FUNCTION_BLOCK FB_TaskMoveZ_creator IMPLEMENTS InterfaceTaskCreator
VAR_INPUT
END_VAR
VAR_OUTPUT
END_VAR
VAR
	_p				: MC_LREAL;
	_v				: MC_LREAL;
	_a				: MC_LREAL;
	_d				: MC_LREAL;
	_j				: MC_LREAL;
	_mover			: REFERENCE TO MC_PlanarMover;
END_VAR

{warning 'add method implementation '}
METHOD create_future : jobmgmt.InterfaceFuture
VAR_INPUT
	future_name	: STRING;
END_VAR
VAR
	_p_future : POINTER TO FB_TaskMoveZ;
END_VAR
_p_future := __NEW(FB_TaskMoveZ);
_p_future^.mover REF= _mover;
_p_future^.future_name := future_name;
_p_future^.set_dynamics(_v,_a,_d,_j);
_p_future^.set_target_position(_p);
create_future := _p_future^;
END_METHOD

{warning 'add method implementation '}
METHOD destroy_future : InterfaceFuture
VAR_INPUT
	future	: jobmgmt.InterfaceFuture;
END_VAR
VAR
	_p_future : POINTER TO FB_TaskMoveZ;
END_VAR
IF __QUERYPOINTER(future, _p_future) THEN
	__DELETE(_p_future);
	IF _p_future = 0  THEN
		destroy_future := 0;
	END_IF
END_IF
END_METHOD

METHOD FB_init : BOOL
VAR_INPUT
	bInitRetains : BOOL; // if TRUE, the retain variables are initialized (warm start / cold start)
	bInCopyCode : BOOL;  // if TRUE, the instance afterwards gets moved into the copy code (online change)
	mover : REFERENCE TO MC_PlanarMover;
END_VAR
_mover REF= mover;
END_METHOD

METHOD set_dynamics : BOOL
VAR_INPUT
	v: MC_LREAL;
	a: MC_LREAL;
	d: MC_LREAL;
	j: MC_LREAL;
END_VAR
_v := v;
_a := a;
_d := d;
_j := j;
set_dynamics := TRUE;
END_METHOD

METHOD set_target_position : BOOL
VAR_INPUT
	z: LREAL;
END_VAR
_p := z;

set_target_position := TRUE;
END_METHOD

END_FUNCTION_BLOCK

(* stored: Version 1.1.0.1, ProductVersion 3.1.4024.12
   POU FB_TaskMoveZ_creator: Id {e1791e19-2621-4797-9a66-d31f7ec5a96b}, SpecialFunc None
   Method create_future: Id {5f5bf45a-f602-460e-9f12-296f268b8061}
   Method destroy_future: Id {0d98a547-8809-492a-b434-6dbf4468ad9a}
   Method FB_init: Id {cf946c34-faed-4236-b6fe-e74f284cb00c}
   Method set_dynamics: Id {3af1285f-54b0-451c-8684-3ecd9d613791}
   Method set_target_position: Id {0f49d619-1b16-4058-90d9-bc633dae23c4} *)
